TYPE TFDatiDaLineaAPal :
STRUCT

	LastraProntaSuPrelievo 		AT %I* : BOOL;//Lastra pronta sul prelievo i-esimo
	LastraPrelevataDaPrelievo  	AT %Q* : BOOL;//Lastra prelevata da pallettizzatore
	DatiLastraSuPrelievo		AT %I* : TFSlab;
	StatoPrelievo				AT %I* : INT;//Stato rulliera prelievo
	StatoPalettizzatore			AT %Q* : INT;//STtao pallettizzatore
	PinzaInIngombro				AT %Q* : BOOL; //Pinza in ongombro
	
END_STRUCT
END_TYPE

(* stored: Version 1.1.0.1, ProductVersion 3.1.4024.9
   DUT TFDatiDaLineaAPal: Id {37a08e06-5cdd-46e7-8131-6cb92c6629f7} *)
